{attribute 'qualified_only'}
VAR_GLOBAL
	bStart AT%Q*	:BOOL;
END_VAR

(* stored: Version 1.1.0.1, ProductVersion 3.1.4026.6
   GVL SignalOut: Id {681f314d-36ea-443c-8345-c3a7de79dcfa} *)
